FUNCTION_BLOCK FB_HMIBase
VAR
	status : ST_HMIStatus;
	configs : ST_HMIConfiguration;
	cmd : ST_HMICommand;
END_VAR

PROPERTY P_Command : ST_HMICommand
GET
END_GET
SET
END_SET
END_PROPERTY

PROPERTY P_Configuration : ST_HMIConfiguration
GET
END_GET
SET
END_SET
END_PROPERTY

PROPERTY P_Status : ST_HMIStatus
GET
END_GET
SET
END_SET
END_PROPERTY

END_FUNCTION_BLOCK

(* stored: Version 1.1.0.1
   POU FB_HMIBase: Id {cccc0bf6-9b64-42bd-b0ca-ff96aa8733e1}, SpecialFunc None
   Property P_Command: Id {38295d4b-cf4d-4043-84fe-a4c04f115626}
   Get Get: Id {9b131594-f8fe-44c4-8bf9-083acf6f22cc}
   Set Set: Id {b2d54d4d-2213-4994-9d02-523a074ae486}
   Property P_Configuration: Id {31ae0e68-4b5e-42f8-9f49-670536860f46}
   Get Get: Id {06472986-6a69-49ed-9c99-19dfabc741dc}
   Set Set: Id {9e1842d2-0fe7-4807-9c85-b2d7770a50c1}
   Property P_Status: Id {f5c47947-7d01-41d6-834a-78421613186a}
   Get Get: Id {10f29e8a-bebe-4e99-ab24-dc1bfc325cde}
   Set Set: Id {a4780232-334c-4510-a907-cfe7552427cb} *)
